FUNCTION TryConvert_USINT_TO_TIME : BOOL
VAR_INPUT
	in : USINT;
	out : REFERENCE TO TIME;
END_VAR

out := USINT_TO_TIME(in);
TryConvert_USINT_TO_TIME := TRUE;

END_FUNCTION

(* stored: Version 1.1.0.1, ProductVersion 3.1.4024.12
   POU TryConvert_USINT_TO_TIME: Id {f176bf1d-5816-40ca-afb3-424aeeff9b69}, SpecialFunc None *)
